FUNCTION ASSEMBLE_BYTE_FROM_BOOLS (* this Function combines the 8 BOOLS to a BYTE *)
  (* Standard: 61499-1; Description: Copyright (c) 2024 HR Agrartechnik GmbH This program and the accompanying materials are made available under the terms of the Eclipse Public License 2.0 which is available at https://www.eclipse.org/legal/epl-2.0/ SPDX-License-Identifier: EPL-2.0 *)
  (* Version 3.0, 2025-04-14, Patrick Aigner, changed package *)
  (* Version 1.1, 2024-07-28, Moritz Ortmeier, HR Agrartechnik, rename Function and change Input/Output Variables *)
  (* Version 1.0, 2024-02-22, Franz H??pfinger, HR Agrartechnik, initial Implementation *)
  PACKAGE eclipse4diac::utils::assembling;
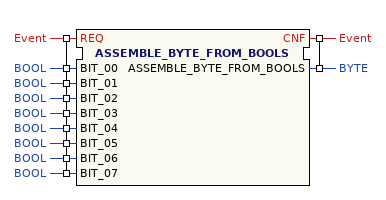
  EVENT_INPUT
    REQ WITH BIT_00, BIT_01, BIT_02, BIT_03, BIT_04, BIT_05, BIT_06, BIT_07;
  END_EVENT
  EVENT_OUTPUT
    CNF WITH ASSEMBLE_BYTE_FROM_BOOLS;
  END_EVENT
  VAR_INPUT
    BIT_00 : BOOL;
    BIT_01 : BOOL;
    BIT_02 : BOOL;
    BIT_03 : BOOL;
    BIT_04 : BOOL;
    BIT_05 : BOOL;
    BIT_06 : BOOL;
    BIT_07 : BOOL;
  END_VAR
  VAR_OUTPUT
    ASSEMBLE_BYTE_FROM_BOOLS : BYTE;
  END_VAR
  BODY IN ST:
(* this Function combines the 8 BOOLS to a BYTE *)
FUNCTION ASSEMBLE_BYTE_FROM_BOOLS : BYTE

VAR_INPUT
	BIT_00 : BOOL;
	BIT_01 : BOOL;
	BIT_02 : BOOL;
	BIT_03 : BOOL;
	BIT_04 : BOOL;
	BIT_05 : BOOL;
	BIT_06 : BOOL;
	BIT_07 : BOOL;
END_VAR

ASSEMBLE_BYTE_FROM_BOOLS.%X0 := BIT_00;
ASSEMBLE_BYTE_FROM_BOOLS.%X1 := BIT_01;
ASSEMBLE_BYTE_FROM_BOOLS.%X2 := BIT_02;
ASSEMBLE_BYTE_FROM_BOOLS.%X3 := BIT_03;
ASSEMBLE_BYTE_FROM_BOOLS.%X4 := BIT_04;
ASSEMBLE_BYTE_FROM_BOOLS.%X5 := BIT_05;
ASSEMBLE_BYTE_FROM_BOOLS.%X6 := BIT_06;
ASSEMBLE_BYTE_FROM_BOOLS.%X7 := BIT_07;

END_FUNCTION
  END_BODY
END_FUNCTION
